FUNCTION_BLOCK RefactoredDSControl (* Composite Function Block Type *)
  (* Standard: 61499-2 *)
  (* Version 0.0, 2/9/2018, Sandeep Patil, nxtControl GmbH, template *)
  PACKAGE Main;
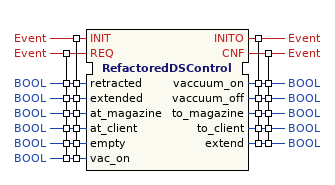
  EVENT_INPUT
    INIT WITH retracted, extended, at_magazine, at_client, empty, vac_on; (* Initialization Request *)
    REQ WITH retracted, extended, at_magazine, at_client, empty, vac_on; (* Normal Execution Request *)
  END_EVENT
  EVENT_OUTPUT
    INITO WITH vaccuum_on, vaccuum_off, to_magazine, to_client, extend; (* Initialization Confirm *)
    CNF WITH vaccuum_on, vaccuum_off, to_magazine, to_client, extend; (* Execution Confirmation *)
  END_EVENT
  VAR_INPUT
    retracted : BOOL;
    extended : BOOL;
    at_magazine : BOOL; (* Input event qualifier *)
    at_client : BOOL;
    empty : BOOL; (* Input event qualifier *)
    vac_on : BOOL;
  END_VAR
  VAR_OUTPUT
    vaccuum_on : BOOL; (* Output event qualifier *)
    vaccuum_off : BOOL;
    to_magazine : BOOL;
    to_client : BOOL;
    extend : BOOL; (* Output event qualifier *)
  END_VAR
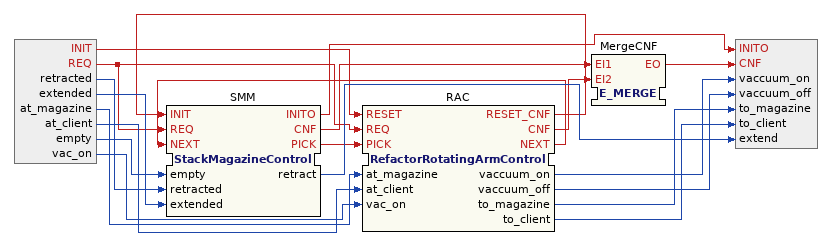
  FBS
    RAC : RefactorRotatingArmControl;
    SMM : StackMagazineControl;
    MergeCNF : E_MERGE;
  END_FBS
  EVENT_CONNECTIONS
    INIT TO RAC.RESET;
    REQ TO SMM.REQ;
    SMM.CNF TO MergeCNF.EI1;
    RAC.CNF TO MergeCNF.EI2;
    MergeCNF.EO TO CNF;
    REQ TO RAC.REQ;
    SMM.PICK TO RAC.PICK;
    RAC.NEXT TO SMM.NEXT;
    RAC.RESET_CNF TO SMM.INIT;
    SMM.INITO TO INITO;
  END_CONNECTIONS
  DATA_CONNECTIONS
    empty TO SMM.empty;
    retracted TO SMM.retracted;
    extended TO SMM.extended;
    at_magazine TO RAC.at_magazine;
    at_client TO RAC.at_client;
    RAC.to_magazine TO to_magazine;
    RAC.to_client TO to_client;
    SMM.retract TO extend;
    vac_on TO RAC.vac_on;
    RAC.vaccuum_on TO vaccuum_on;
    RAC.vaccuum_off TO vaccuum_off;
  END_CONNECTIONS
END_FUNCTION_BLOCK
